Staubli VAL3: setItem.pgx

public program setItem(string x_sItem, string& x_sId[])
  local num l_nSize
begin
  // set the ITEM name
  saveInOut:dInput[x_sId].sName=x_sItem
end
